{attribute 'TcGenerated'}
// This function has been automatically generated from the project information.
VAR_GLOBAL CONSTANT
    {attribute 'const_non_replaced'}
    {attribute 'linkalways'}
    stLibVersion_lcls_plc_crix_vac : ST_LibVersion := (iMajor := 2, iMinor := 1, iBuild := 0, iRevision := 0, sVersion := '2.1.0');
END_VAR

(* stored: Version 1.1.0.1, ProductVersion 3.1.4022.18
   GVL Global_Version: Id 7e75386b-d922-4cf2-8d8e-317ac978dfcf *)
